Staubli VAL3: Init.pgx

program Init()
  local num l_ni
begin
  //
  bUserRefresh=bListRefresh=true
  //
  bExit=false
  //
  call readFileList(sFolder,sFileList)
  call selectFile(sDeli,sFileList)
  //

end
